(*********************************** G.D S.p.A. - Technical Department ***********************************
============= PROGRAM INFO ============
FOLDER:             TBD
MACHINES INVOLVED:  TBD 

============= DESCRIPTION =============
csp main interface program

============= REVISIONS ===============
Date		Version	 	Author      	Description             
----------	-------		------------  	--------------------------------------------
2019/09/27 	0000.00	 	M.Grasso		Creation of the PRG

**********************************************************************************************************)
PROGRAM _csp_case_loader_normal
VAR
END_VAR

(* CASE *)
	(* LOADER *)
		(* GUIDE *)
		csp_case_loader_guide();
		(* SENSORS *)
		csp_case_loader_sensors();

END_PROGRAM

(* stored: Version 1.1.0.1, ProductVersion 3.1.4024.3
   POU _csp_case_loader_normal: Id {c928abf6-1305-43f1-bf4f-7fd8488cebd6}, SpecialFunc None *)
